FUNCTION_BLOCK CarriageModelView
  (* Standard: 61499-2 *)
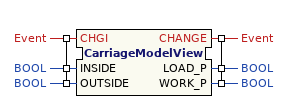
  EVENT_INPUT
    CHGI WITH INSIDE, OUTSIDE;
  END_EVENT
  EVENT_OUTPUT
    CHANGE WITH LOAD_P, WORK_P;
  END_EVENT
  VAR_INPUT
    INSIDE : BOOL;
    OUTSIDE : BOOL;
  END_VAR
  VAR_OUTPUT
    LOAD_P : BOOL;
    WORK_P : BOOL;
  END_VAR
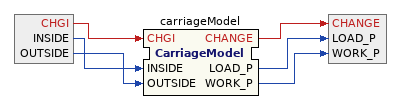
  FBS
    carriageModel : CarriageModel;
  END_FBS
  EVENT_CONNECTIONS
    CHGI TO carriageModel.CHGI;
    carriageModel.CHANGE TO CHANGE;
  END_CONNECTIONS
  DATA_CONNECTIONS
    carriageModel.LOAD_P TO LOAD_P;
    carriageModel.WORK_P TO WORK_P;
    INSIDE TO carriageModel.INSIDE;
    OUTSIDE TO carriageModel.OUTSIDE;
  END_CONNECTIONS
END_FUNCTION_BLOCK
